FUNCTION_BLOCK Q_SelectActiveWorkingSet (* Command Select Active Working Set( Part 6 - F.64 ) *)
  (* Standard: ISO 11783-6; Description: see Description Tab *)
  (* Version 1.0, 2022-07-08, franz *)
  (* Documentation:
  Command Select Active Working Set( Part 6 - F.64 )
   This command is used by the currently active Working Set to request that the VT select a new active Working Set. This message is available in VT version 6 and later.
   param[in] {NAMEofWorkingSetMasterForDesiredWorkingSet,  const uint8_t *}
   Iso NAME of the new active working set
   Return Values: 
   int16_t
    - VT_E_NO_ERR (0) - OK
   - VT_E_OVERFLOW (-6) - buffer overflow
   - VT_E_NOACT (-8) - Command not possible in current state
   - VT_E_NO_INSTANCE (-21) - No VT client available
   - VT_E_ISO_INSTANCE_INVALID (-129) - Identifier for instance (connection) invalid
   - VT_E_NOT_ALVIE (-130) - Identifier for instance valid, but VT Dead.
  *)
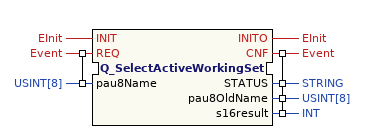
  EVENT_INPUT
    INIT : EInit; (* Service Initialization *)
    REQ WITH pau8Name; (* Service Request *)
  END_EVENT
  EVENT_OUTPUT
    INITO : EInit; (* Initialization Confirm *)
    CNF WITH STATUS, pau8OldName, s16result; (* Confirmation of Requested Service *)
  END_EVENT
  VAR_INPUT
    pau8Name : ARRAY [0..7] OF USINT; (* Iso NAME of the new active working set *)
  END_VAR
  VAR_OUTPUT
    STATUS : STRING; (* Service Status *)
    pau8OldName : ARRAY [0..7] OF USINT; (* Old value of Visible *)
    s16result : INT; (* retval see description *)
  END_VAR
END_FUNCTION_BLOCK
